FUNCTION_BLOCK FB_TankController IMPLEMENTS I_TankController


VAR_IN_OUT
	stTank : ST_Tank;
END_VAR
VAR
	eState : E_TankState;
END_VAR


IF __ISVALIDREF(stTank) THEN
	eState := stTank.eState;
	CheckSafety();
	CASE eState OF
		E_TankState.Idle:
		
		IF NOT stTank.bAlarm THEN
			stTank.eState := E_TankState.Filling;
		END_IF
		E_TankState.Filling:
		
		IF NOT stTank.bAlarm THEN
			stTank.eState := E_TankState.Filling;
		END_IF
		E_TankState.Processing:
		
		E_TankState.Dispensing:
		
		E_TankState.Cooling:
		
		E_TankState.Alarm:
	END_CASE

	
END_IF

{warning 'add method implementation '}
METHOD ApplyCooling : BOOL
IF stTank.bAlarm THEN
	F_CoolTank(stTank);
END_IF
END_METHOD

{warning 'add method implementation '}
METHOD CheckSafety : BOOL
IF F_CheckAlarm( pTank := ADR(stTank) ) THEN
	stTank.bAlarm := TRUE;
END_IF
END_METHOD

METHOD TransferChemical : BOOL
VAR_INPUT
END_VAR
END_METHOD

END_FUNCTION_BLOCK

(* stored: Version 1.1.0.1, ProductVersion 3.1.4024.16
   POU FB_TankController: Id {bd5580ac-b1f3-4fa5-92f5-0a91a9517670}, SpecialFunc None
   Method ApplyCooling: Id {41f3f916-3681-4c60-b39a-5ab8cb364b13}
   Method CheckSafety: Id {dee3a59f-b24f-4a00-879d-a7220b0c9cf6}
   Method TransferChemical: Id {f6ebb983-a058-4a80-a535-bcd72625ef5a} *)
